FUNCTION_BLOCK EffluentCdt (* CAT Function Block Type *)
  (* Standard: 61499-2 *)
  (* Version 0.0, 6/7/2026, Schneider Electric, template *)
  PACKAGE SE.Nereda;
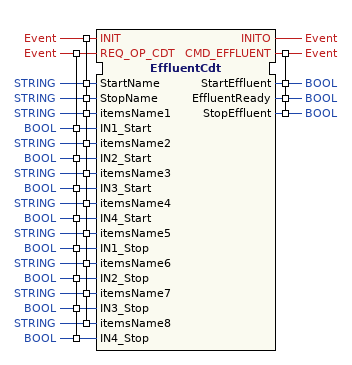
  EVENT_INPUT
    INIT WITH itemsName1, itemsName2, itemsName3, itemsName4, itemsName5, itemsName6, itemsName7, itemsName8, StartName, StopName;
    REQ_OP_CDT WITH IN1_Start, IN2_Start, IN3_Start, IN4_Start, IN1_Stop, IN2_Stop, IN3_Stop, IN4_Stop; (* Normal Execution Request *)
  END_EVENT
  EVENT_OUTPUT
    INITO;
    CMD_EFFLUENT WITH StartEffluent, EffluentReady, StopEffluent; (* Input changed *)
  END_EVENT
  VAR_INPUT
    StartName : STRING;
    StopName : STRING;
    itemsName1 : STRING;
    IN1_Start : BOOL; (* Argument *)
    itemsName2 : STRING;
    IN2_Start : BOOL; (* Argument *)
    itemsName3 : STRING;
    IN3_Start : BOOL; (* Argument *)
    itemsName4 : STRING;
    IN4_Start : BOOL; (* Argument *)
    itemsName5 : STRING;
    IN1_Stop : BOOL; (* Argument *)
    itemsName6 : STRING;
    IN2_Stop : BOOL; (* Argument *)
    itemsName7 : STRING;
    IN3_Stop : BOOL; (* Argument *)
    itemsName8 : STRING;
    IN4_Stop : BOOL; (* Argument *)
  END_VAR
  VAR_OUTPUT
    StartEffluent : BOOL; (* Output value *)
    EffluentReady : BOOL; (* Output value *)
    StopEffluent : BOOL; (* Output value *)
  END_VAR
  (* 01 - FUNCTIONNAL INPUT INTERFACE *)
  (* 05 - LOGIC *)
  (* 02 - FUNCTIONNAL OUTPUT INTERFACE *)
  (* 00 - INITIALIZATION *)
  (* 06 - HMI INTERFACE *)
  (* 03 - FIELD INTERFACE *)
  (* Conditions : IN1_Start =>    'Start Pump - Effluent' IN2_Start =>    'NVPP 001 a-- 011 is Available' IN3_Start =>    'NVPP 001 a-- 014 is Available' IN4_Start =>    'Effluent Pump is Ready' IN1_Stop =>    'Stop Pump - Effluent' IN2_Stop =>    'Hight Hight Level - Calamity' IN3_Stop =>    'Low Level - Effluent' IN4_Stop =>    ---- *)
  FBS
    StartCdts : AND_150A6959DE81880FD; {SET_ATTRIBUTE(Configuration.GenericFBType.InterfaceParams, Runtime.Standard#CNT:=5;OUT:BOOL)}
    encodeB1 : VALFORMAT_95B1C22C7F49B890(FORMAT := '%s%s%s%s'); {SET_ATTRIBUTE(Configuration.GenericFBType.InterfaceParams, Runtime.Standard#I:=4;VALUE${I$}:INT,INT,INT,INT)}
    encodeB2 : VALFORMAT_95B1C22C7F49B890(FORMAT := '%s%s%s%s'); {SET_ATTRIBUTE(Configuration.GenericFBType.InterfaceParams, Runtime.Standard#I:=4;VALUE${I$}:INT,INT,INT,INT)}
    StartCdtsSmooth : boolValueChanged;
    IThis : EffluentCdt_HMI(QI := TRUE);
    StopCdtsSmooth : boolValueChanged;
    CMD : E_MERGE_4;
    StopCdts : OR_169B00D031196E7C4; {SET_ATTRIBUTE(Configuration.GenericFBType.InterfaceParams, Runtime.Standard#CNT:=4;OUT:BOOL)}
    ReadyCdtsSmooth : boolValueChanged;
    ReadyCdts : AND_150A6959DE81880FD; {SET_ATTRIBUTE(Configuration.GenericFBType.InterfaceParams, Runtime.Standard#CNT:=5;OUT:BOOL)}
    NoLowLow : NOT_42C76073DCEB1A7A; {SET_ATTRIBUTE(Configuration.GenericFBType.InterfaceParams, Runtime.Standard#CNT:=1;OUT${CNT$}:BOOL)}
    NoHighHighCalamity : NOT_42C76073DCEB1A7A; {SET_ATTRIBUTE(Configuration.GenericFBType.InterfaceParams, Runtime.Standard#CNT:=1;OUT${CNT$}:BOOL)}
    NOT_Stop : NOT_42C76073DCEB1A7A; {SET_ATTRIBUTE(Configuration.GenericFBType.InterfaceParams, Runtime.Standard#CNT:=1;OUT${CNT$}:BOOL)}
    OverrideValues : OverrideV;
    STR2INT1 : STR2INT;
    STR2INT2 : STR2INT;
    BOOL2INT1 : BOOL2INT_4;
    BOOL2INT2 : BOOL2INT_4;
  END_FBS
  EVENT_CONNECTIONS
    REQ_OP_CDT TO StopCdts.REQ;
    StartCdtsSmooth.CNF TO ReadyCdtsSmooth.REQ;
    NoLowLow.CNF TO ReadyCdts.REQ;
    NoHighHighCalamity.CNF TO NoLowLow.REQ;
    INIT TO IThis.7D98611DC811A4F7;
    IThis.8A8403C8DB481D6C TO IThis.6D29BCFC45D76FE3;
    IThis.8A8403C8DB481D6C TO IThis.A665539B906F6DBA;
    IThis.8A8403C8DB481D6C TO INITO;
    StopCdts.CNF TO NOT_Stop.REQ;
    NOT_Stop.CNF TO StartCdts.REQ;
    ReadyCdtsSmooth.CNF TO StopCdtsSmooth.REQ;
    StartCdts.CNF TO NoHighHighCalamity.REQ;
    BOOL2INT1.6FC99A5BD1C38561 TO encodeB1.REQ;
    encodeB1.CNF TO STR2INT1.DD5870AA881150BB;
    STR2INT1.6FC99A5BD1C38561 TO BOOL2INT2.DD5870AA881150BB;
    BOOL2INT2.6FC99A5BD1C38561 TO encodeB2.REQ;
    ReadyCdts.CNF TO OverrideValues.806431ABD5E78883;
    IThis.60A7F243DF4A4B8D TO OverrideValues.806431ABD5E78883;
    OverrideValues.B861589364FF8D2A TO StartCdtsSmooth.REQ;
    StopCdtsSmooth.CNF TO BOOL2INT1.DD5870AA881150BB;
    StopCdtsSmooth.CHD TO CMD.EI2;
    encodeB2.CNF TO STR2INT2.DD5870AA881150BB;
    STR2INT2.6FC99A5BD1C38561 TO IThis.6D29BCFC45D76FE3;
    StartCdtsSmooth.CHD TO CMD.EI1;
    ReadyCdtsSmooth.CHD TO CMD.EI3;
    CMD.EO TO CMD_EFFLUENT;
  END_CONNECTIONS
  DATA_CONNECTIONS
    IN1_Stop TO StopCdts.IN1;
    IN2_Stop TO StopCdts.IN2;
    IN3_Stop TO StopCdts.IN3;
    IN4_Stop TO StopCdts.IN4;
    StartCdtsSmooth.Output TO StartEffluent;
    StopCdtsSmooth.Output TO StopEffluent;
    ReadyCdtsSmooth.Output TO EffluentReady;
    NoLowLow.OUT1 TO ReadyCdts.IN1;
    IN2_Start TO ReadyCdts.IN2;
    IN3_Start TO ReadyCdts.IN3;
    IN4_Start TO ReadyCdts.IN4;
    NoHighHighCalamity.OUT1 TO ReadyCdts.IN5;
    IN2_Stop TO NoHighHighCalamity.IN1;
    StartCdtsSmooth.Output TO IThis.52F65A7B68D385BC;
    ReadyCdtsSmooth.Output TO IThis.C73BA7FBEF416DF3;
    StopCdtsSmooth.Output TO IThis.41ACDF6E671E7491;
    StartName TO IThis.5F8F361E80D292F1;
    StopName TO IThis.DC3E27EDA0187D96;
    itemsName1 TO IThis.74E1E0951D70046E;
    itemsName2 TO IThis.EE9470BA0350B131;
    itemsName3 TO IThis.EDAEBE4CEBDB9AE9;
    itemsName4 TO IThis.521EB392A39EAFAC;
    itemsName5 TO IThis.882EBDE88CE34770;
    itemsName6 TO IThis.CFFC3D70D2D95759;
    itemsName7 TO IThis.FEED97F6C5CA5C81;
    itemsName8 TO IThis.7E2A6F1CECD5D852;
    StopCdts.OUT TO NOT_Stop.IN1;
    IN1_Start TO StartCdts.IN1;
    IN2_Start TO StartCdts.IN2;
    IN3_Start TO StartCdts.IN3;
    IN4_Start TO StartCdts.IN4;
    NOT_Stop.OUT1 TO StartCdts.IN5;
    IThis.2527FEE561F0F361 TO OverrideValues.801967BDFA8F77B6;
    StartCdts.OUT TO OverrideValues.53EE5823BC68BC38;
    ReadyCdts.OUT TO OverrideValues.531474AB7BB2BE86;
    StopCdts.OUT TO OverrideValues.272BD6D99E89DB2E;
    IThis.4736FE9FD6BAE8DC TO OverrideValues.F257BF6AA9E98D5A;
    IThis.6E91CA2C8977A6A0 TO OverrideValues.C73C44DF80BC8DC6;
    IThis.7DAEED1278D5C638 TO OverrideValues.A8FE9F00BB619032;
    OverrideValues.4B7E902E80034964 TO StartCdtsSmooth.Input;
    OverrideValues.FDAA14F9B1820A36 TO ReadyCdtsSmooth.Input;
    OverrideValues.F25E94E81E907B48 TO StopCdtsSmooth.Input;
    IN4_Start TO BOOL2INT1.4573FC8F228EB71D;
    IN3_Start TO BOOL2INT1.DF8224FEB3446E92;
    IN2_Start TO BOOL2INT1.F547CEFAFDE5D422;
    IN1_Start TO BOOL2INT1.25941BC08BA9FF7D;
    BOOL2INT1.A6DEF5F9C27C1848 TO encodeB1.VALUE1;
    BOOL2INT1.515A2E3BB78F58C7 TO encodeB1.VALUE2;
    BOOL2INT1.FCA64FB4B13F606F TO encodeB1.VALUE3;
    BOOL2INT1.740A810221DABFBE TO encodeB1.VALUE4;
    encodeB1.RESULT TO STR2INT1.4573FC8F228EB71D;
    STR2INT1.A6DEF5F9C27C1848 TO IThis.9CD6AD33A52FBF26;
    BOOL2INT2.740A810221DABFBE TO encodeB2.VALUE4;
    BOOL2INT2.FCA64FB4B13F606F TO encodeB2.VALUE3;
    BOOL2INT2.515A2E3BB78F58C7 TO encodeB2.VALUE2;
    BOOL2INT2.A6DEF5F9C27C1848 TO encodeB2.VALUE1;
    IN4_Stop TO BOOL2INT2.4573FC8F228EB71D;
    IN3_Stop TO BOOL2INT2.DF8224FEB3446E92;
    IN2_Stop TO BOOL2INT2.F547CEFAFDE5D422;
    IN1_Stop TO BOOL2INT2.25941BC08BA9FF7D;
    encodeB2.RESULT TO STR2INT2.4573FC8F228EB71D;
    STR2INT2.A6DEF5F9C27C1848 TO IThis.CC812AEED2D2840D;
    IN3_Stop TO NoLowLow.IN1;
  END_CONNECTIONS
END_FUNCTION_BLOCK
